(* Logix 5000 project; controller Safety vendor 1 type 14 code 86 rev 19.11; software revision 19.01; part 3 of 17 *)
(* tags used below, declared in another part *)
   MCC2_IO : UDT_CardSts[32];   // MCC2 Point I/O
   MCC2_IOSts_Flt : BOOL;   // MCC2 Point IO Module Fault ( 1= Faulted)
   MCC3_IO : UDT_CardSts[32];   // MCC3 Point I/O
   MCC3_IOSts_Flt : BOOL;   // MCC3 Point IO Module Fault ( 1= Faulted)
   MCC4_IO : UDT_CardSts[32];   // MCC4 Point I/O
   MCC4_IOSts_Flt : BOOL;   // MCC-4 Point IO Module Fault ( 1= Faulted)
   MCC5_IO : UDT_CardSts[32];   // MCC5 Point I/O
   MCC5_IOSts_Flt : BOOL;   // MCC-5 Point IO Module Fault ( 1= Faulted)
   OS11_IO : UDT_CardSts[32];   // OS11 Point I/O
   OS11_IOSts_Flt : BOOL;   // OS11 Point IO Module Fault ( 1= Faulted)
   OS13_IO : UDT_CardSts[32];   // OS13 Point I/O
   OS13_IOSts_Flt : BOOL;   // OS13 Point IO Module Fault ( 1= Faulted)
   OS14_IO : UDT_CardSts[32];   // OS14 Point I/O
   OS14_IOSts_Flt : BOOL;   // OS14 Point IO Module Fault ( 1= Faulted)
   OS15_IO : UDT_CardSts[32];   // OS15 Point I/O
   OS15_IOSts_Flt : BOOL;   // OS15 Point IO Module Fault ( 1= Faulted)
   OS16_IO : UDT_CardSts[32];   // OS16 Point I/O
   OS16_IOSts_Flt : BOOL;   // OS16 Point IO Module Fault ( 1= Faulted)
   OS1_IO : UDT_CardSts[32];   // OS1 Point I/O
   OS1_IOSts_Flt : BOOL;   // OS1 Point IO Module Fault ( 1= Faulted)
   OS2_IO : UDT_CardSts[32];   // OS2 Point I/O
   OS2_IOSts_Flt : BOOL;   // OS2 Point IO Module Fault ( 1= Faulted)
   OS3_IO : UDT_CardSts[32];   // OS3 Point I/O
   OS3_IOSts_Flt : BOOL;   // OS3 Point IO Module Fault ( 1= Faulted)
   OS4N_IO : UDT_CardSts[32];   // OS4N Point I/O
   OS4N_IOSts_Flt : BOOL;   // OS4N Point IO Module Fault ( 1= Faulted)
   OS4S_IO : UDT_CardSts[32];   // OS4S Point I/O
   OS4S_IOSts_Flt : BOOL;   // OS4S Point IO Module Fault ( 1= Faulted)
   OS5_IO : UDT_CardSts[32];   // OS5 Point I/O
   OS5_IOSts_Flt : BOOL;   // OS5 Point IO Module Fault ( 1= Faulted)
   OS6_IO : UDT_CardSts[32];   // OS6 Point I/O
   OS6_IOSts_Flt : BOOL;   // OS6 Point IO Module Fault ( 1= Faulted)
   OS8_IO : UDT_CardSts[32];   // OS8 Point I/O
   OS8_IOSts_Flt : BOOL;   // OS8 Point IO Module Fault ( 1= Faulted)
   OS9_IO : UDT_CardSts[32];   // OS9 Point I/O
   OS9_IOSts_Flt : BOOL;   // OS9 Point IO Module Fault ( 1= Faulted)
   Rem_ModFlts : DINT;   // Remote IO Comm Faults
   Sy_ClrFlt : BOOL;   // System Clear Fault
(* CardSts, continued *)

ROUTINE MCC2_IO   (* ladder *)
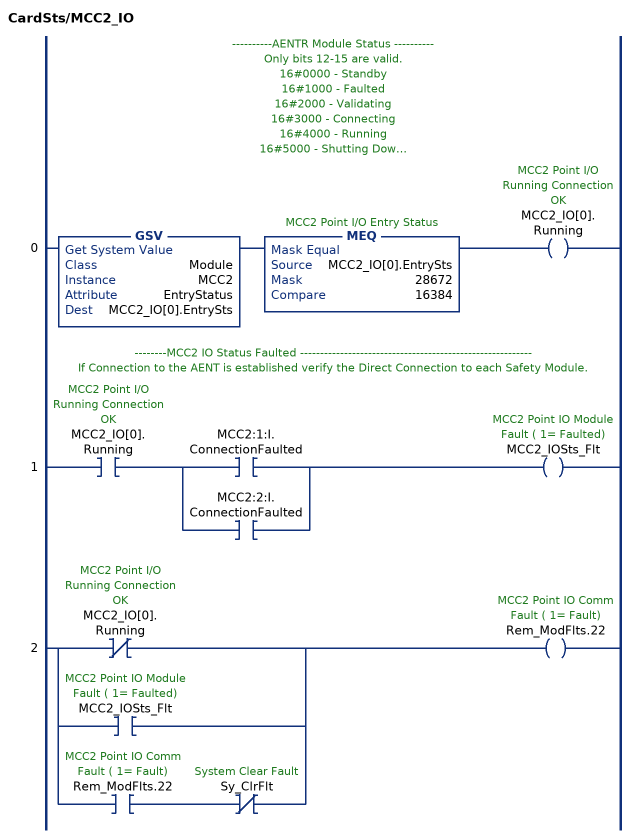
   // ----------AENTR Module Status ----------
   // Only bits 12-15 are valid.
   // 16#0000 - Standby
   // 16#1000 - Faulted
   // 16#2000 - Validating
   // 16#3000 - Connecting
   // 16#4000 - Running
   // 16#5000 - Shutting Down
   // 16#6000 - Inhibited
   // 16#7000 - Waiting
   0: GSV(Module,MCC2,EntryStatus,MCC2_IO[0].EntrySts)MEQ(MCC2_IO[0].EntrySts,28672,16384)OTE(MCC2_IO[0].Running);
   // --------MCC2 IO Status Faulted ----------------------------------------------------------
   // If Connection to the AENT is established verify the Direct Connection to each Safety Module.
   1: XIC(MCC2_IO[0].Running)[XIC(MCC2:1:I.ConnectionFaulted) ,XIC(MCC2:2:I.ConnectionFaulted) ]OTE(MCC2_IOSts_Flt);
   2: [XIO(MCC2_IO[0].Running) ,XIC(MCC2_IOSts_Flt) ,XIC(Rem_ModFlts.22) XIO(Sy_ClrFlt) ]OTE(Rem_ModFlts.22);
END_ROUTINE

ROUTINE MCC3_IO   (* ladder *)
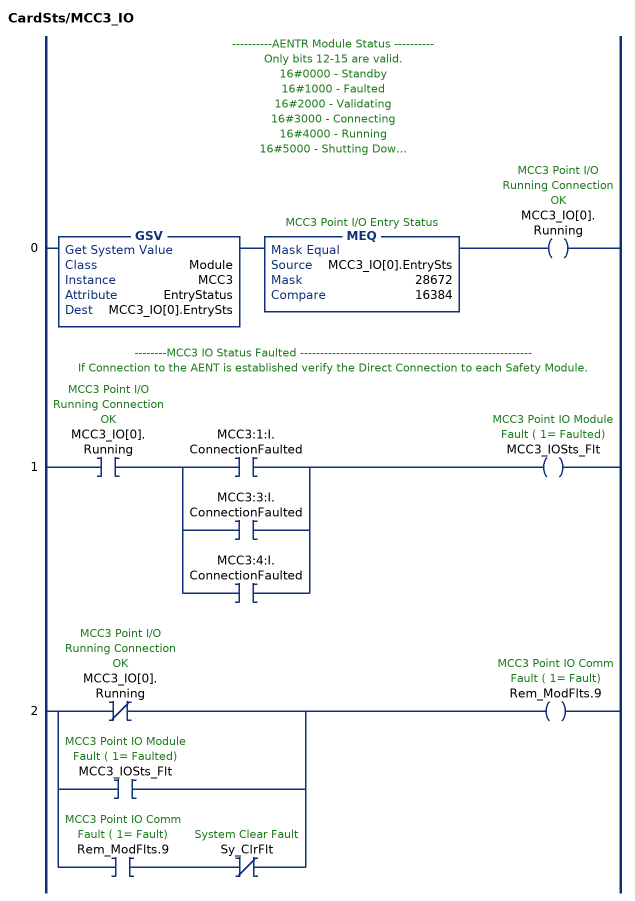
   // ----------AENTR Module Status ----------
   // Only bits 12-15 are valid.
   // 16#0000 - Standby
   // 16#1000 - Faulted
   // 16#2000 - Validating
   // 16#3000 - Connecting
   // 16#4000 - Running
   // 16#5000 - Shutting Down
   // 16#6000 - Inhibited
   // 16#7000 - Waiting
   0: GSV(Module,MCC3,EntryStatus,MCC3_IO[0].EntrySts)MEQ(MCC3_IO[0].EntrySts,28672,16384)OTE(MCC3_IO[0].Running);
   // --------MCC3 IO Status Faulted ----------------------------------------------------------
   // If Connection to the AENT is established verify the Direct Connection to each Safety Module.
   1: XIC(MCC3_IO[0].Running)[XIC(MCC3:1:I.ConnectionFaulted) ,XIC(MCC3:3:I.ConnectionFaulted) ,XIC(MCC3:4:I.ConnectionFaulted) ]OTE(MCC3_IOSts_Flt);
   2: [XIO(MCC3_IO[0].Running) ,XIC(MCC3_IOSts_Flt) ,XIC(Rem_ModFlts.9) XIO(Sy_ClrFlt) ]OTE(Rem_ModFlts.9);
END_ROUTINE

ROUTINE MCC4_IO   (* ladder *)
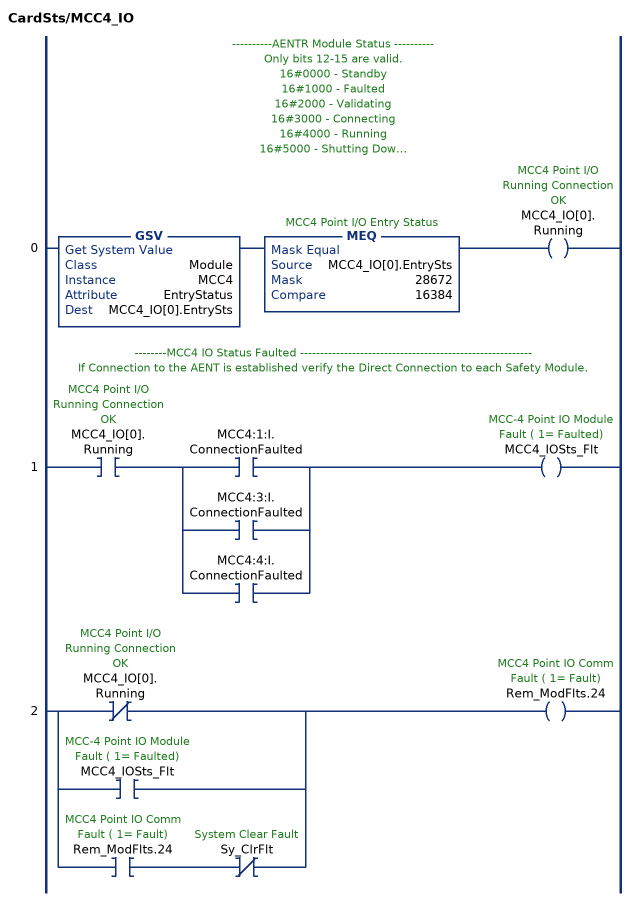
   // ----------AENTR Module Status ----------
   // Only bits 12-15 are valid.
   // 16#0000 - Standby
   // 16#1000 - Faulted
   // 16#2000 - Validating
   // 16#3000 - Connecting
   // 16#4000 - Running
   // 16#5000 - Shutting Down
   // 16#6000 - Inhibited
   // 16#7000 - Waiting
   0: GSV(Module,MCC4,EntryStatus,MCC4_IO[0].EntrySts)MEQ(MCC4_IO[0].EntrySts,28672,16384)OTE(MCC4_IO[0].Running);
   // --------MCC4 IO Status Faulted ----------------------------------------------------------
   // If Connection to the AENT is established verify the Direct Connection to each Safety Module.
   1: XIC(MCC4_IO[0].Running)[XIC(MCC4:1:I.ConnectionFaulted) ,XIC(MCC4:3:I.ConnectionFaulted) ,XIC(MCC4:4:I.ConnectionFaulted) ]OTE(MCC4_IOSts_Flt);
   2: [XIO(MCC4_IO[0].Running) ,XIC(MCC4_IOSts_Flt) ,XIC(Rem_ModFlts.24) XIO(Sy_ClrFlt) ]OTE(Rem_ModFlts.24);
END_ROUTINE

ROUTINE MCC5_IO   (* ladder *)
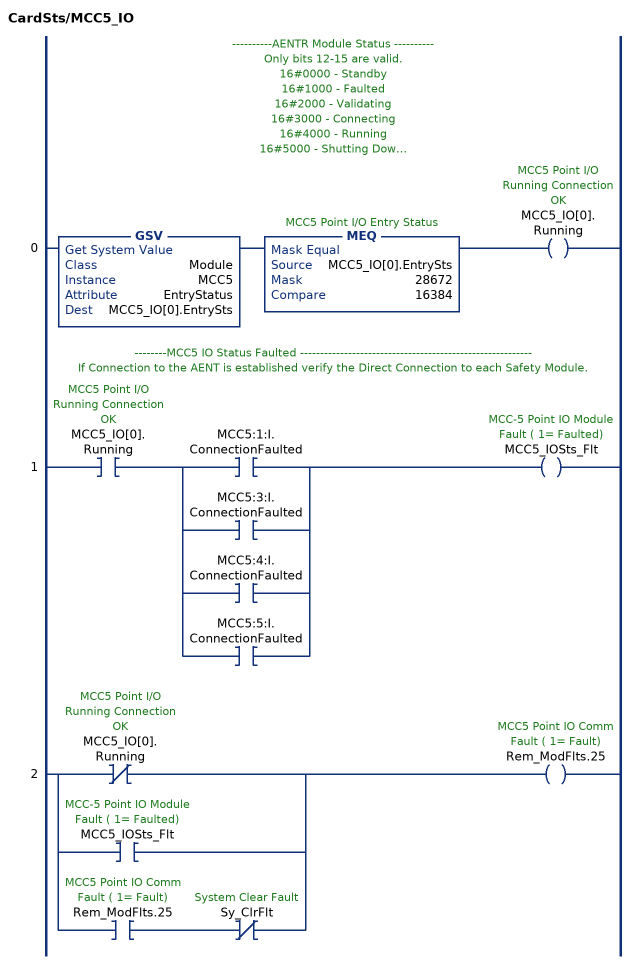
   // ----------AENTR Module Status ----------
   // Only bits 12-15 are valid.
   // 16#0000 - Standby
   // 16#1000 - Faulted
   // 16#2000 - Validating
   // 16#3000 - Connecting
   // 16#4000 - Running
   // 16#5000 - Shutting Down
   // 16#6000 - Inhibited
   // 16#7000 - Waiting
   0: GSV(Module,MCC5,EntryStatus,MCC5_IO[0].EntrySts)MEQ(MCC5_IO[0].EntrySts,28672,16384)OTE(MCC5_IO[0].Running);
   // --------MCC5 IO Status Faulted ----------------------------------------------------------
   // If Connection to the AENT is established verify the Direct Connection to each Safety Module.
   1: XIC(MCC5_IO[0].Running)[XIC(MCC5:1:I.ConnectionFaulted) ,XIC(MCC5:3:I.ConnectionFaulted) ,XIC(MCC5:4:I.ConnectionFaulted) ,XIC(MCC5:5:I.ConnectionFaulted) ]OTE(MCC5_IOSts_Flt);
   2: [XIO(MCC5_IO[0].Running) ,XIC(MCC5_IOSts_Flt) ,XIC(Rem_ModFlts.25) XIO(Sy_ClrFlt) ]OTE(Rem_ModFlts.25);
END_ROUTINE

ROUTINE OS11_IO   (* ladder *)
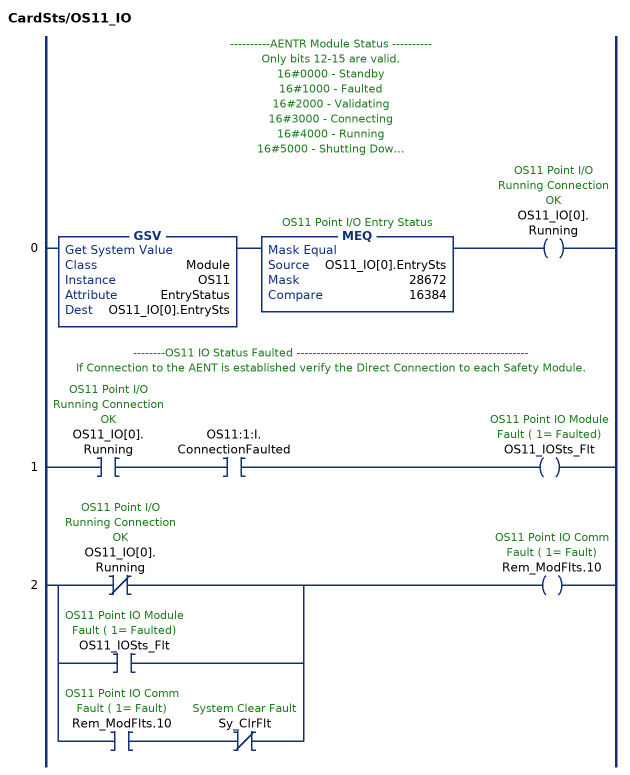
   // ----------AENTR Module Status ----------
   // Only bits 12-15 are valid.
   // 16#0000 - Standby
   // 16#1000 - Faulted
   // 16#2000 - Validating
   // 16#3000 - Connecting
   // 16#4000 - Running
   // 16#5000 - Shutting Down
   // 16#6000 - Inhibited
   // 16#7000 - Waiting
   0: GSV(Module,OS11,EntryStatus,OS11_IO[0].EntrySts)MEQ(OS11_IO[0].EntrySts,28672,16384)OTE(OS11_IO[0].Running);
   // --------OS11 IO Status Faulted ----------------------------------------------------------
   // If Connection to the AENT is established verify the Direct Connection to each Safety Module.
   1: XIC(OS11_IO[0].Running)XIC(OS11:1:I.ConnectionFaulted)OTE(OS11_IOSts_Flt);
   2: [XIO(OS11_IO[0].Running) ,XIC(OS11_IOSts_Flt) ,XIC(Rem_ModFlts.10) XIO(Sy_ClrFlt) ]OTE(Rem_ModFlts.10);
END_ROUTINE

ROUTINE OS13_IO   (* ladder *)
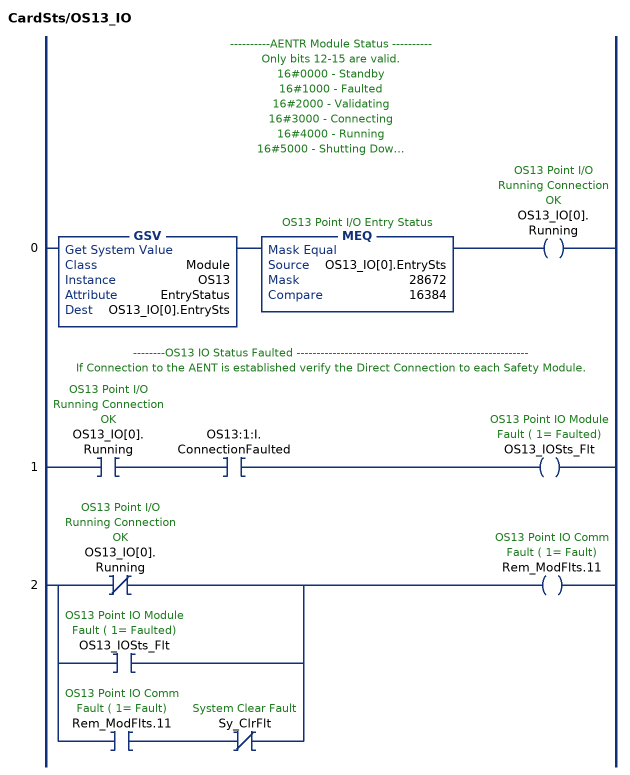
   // ----------AENTR Module Status ----------
   // Only bits 12-15 are valid.
   // 16#0000 - Standby
   // 16#1000 - Faulted
   // 16#2000 - Validating
   // 16#3000 - Connecting
   // 16#4000 - Running
   // 16#5000 - Shutting Down
   // 16#6000 - Inhibited
   // 16#7000 - Waiting
   0: GSV(Module,OS13,EntryStatus,OS13_IO[0].EntrySts)MEQ(OS13_IO[0].EntrySts,28672,16384)OTE(OS13_IO[0].Running);
   // --------OS13 IO Status Faulted ----------------------------------------------------------
   // If Connection to the AENT is established verify the Direct Connection to each Safety Module.
   1: XIC(OS13_IO[0].Running)XIC(OS13:1:I.ConnectionFaulted)OTE(OS13_IOSts_Flt);
   2: [XIO(OS13_IO[0].Running) ,XIC(OS13_IOSts_Flt) ,XIC(Rem_ModFlts.11) XIO(Sy_ClrFlt) ]OTE(Rem_ModFlts.11);
END_ROUTINE

ROUTINE OS14_IO   (* ladder *)
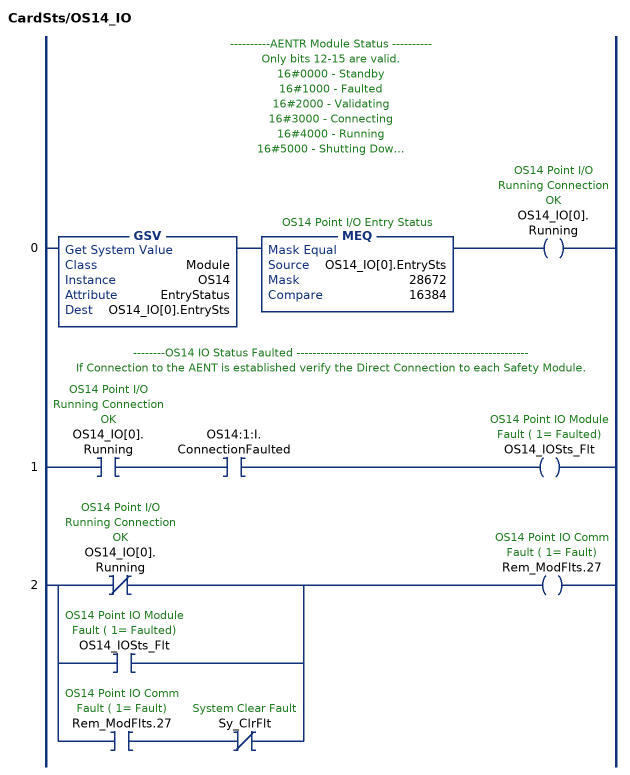
   // ----------AENTR Module Status ----------
   // Only bits 12-15 are valid.
   // 16#0000 - Standby
   // 16#1000 - Faulted
   // 16#2000 - Validating
   // 16#3000 - Connecting
   // 16#4000 - Running
   // 16#5000 - Shutting Down
   // 16#6000 - Inhibited
   // 16#7000 - Waiting
   0: GSV(Module,OS14,EntryStatus,OS14_IO[0].EntrySts)MEQ(OS14_IO[0].EntrySts,28672,16384)OTE(OS14_IO[0].Running);
   // --------OS14 IO Status Faulted ----------------------------------------------------------
   // If Connection to the AENT is established verify the Direct Connection to each Safety Module.
   1: XIC(OS14_IO[0].Running)XIC(OS14:1:I.ConnectionFaulted)OTE(OS14_IOSts_Flt);
   2: [XIO(OS14_IO[0].Running) ,XIC(OS14_IOSts_Flt) ,XIC(Rem_ModFlts.27) XIO(Sy_ClrFlt) ]OTE(Rem_ModFlts.27);
END_ROUTINE

ROUTINE OS15_IO   (* ladder *)
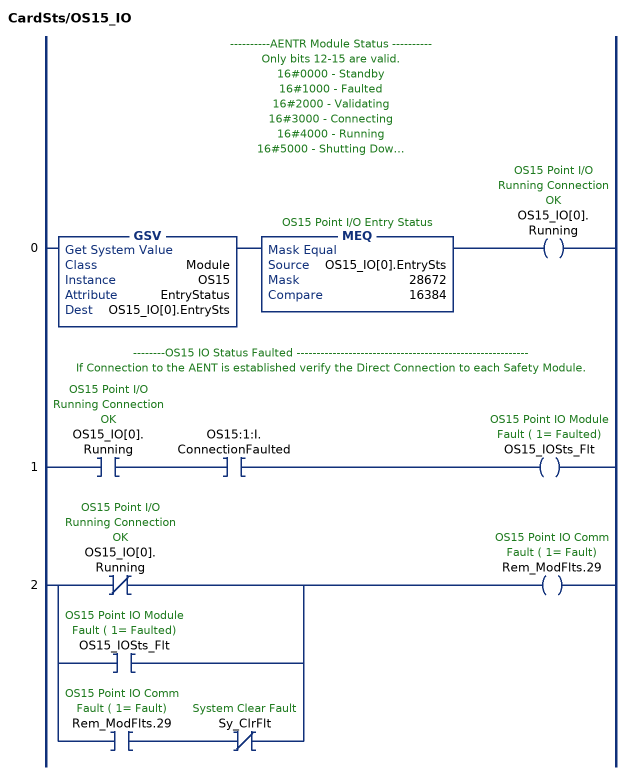
   // ----------AENTR Module Status ----------
   // Only bits 12-15 are valid.
   // 16#0000 - Standby
   // 16#1000 - Faulted
   // 16#2000 - Validating
   // 16#3000 - Connecting
   // 16#4000 - Running
   // 16#5000 - Shutting Down
   // 16#6000 - Inhibited
   // 16#7000 - Waiting
   0: GSV(Module,OS15,EntryStatus,OS15_IO[0].EntrySts)MEQ(OS15_IO[0].EntrySts,28672,16384)OTE(OS15_IO[0].Running);
   // --------OS15 IO Status Faulted ----------------------------------------------------------
   // If Connection to the AENT is established verify the Direct Connection to each Safety Module.
   1: XIC(OS15_IO[0].Running)XIC(OS15:1:I.ConnectionFaulted)OTE(OS15_IOSts_Flt);
   2: [XIO(OS15_IO[0].Running) ,XIC(OS15_IOSts_Flt) ,XIC(Rem_ModFlts.29) XIO(Sy_ClrFlt) ]OTE(Rem_ModFlts.29);
END_ROUTINE

ROUTINE OS16_IO   (* ladder *)
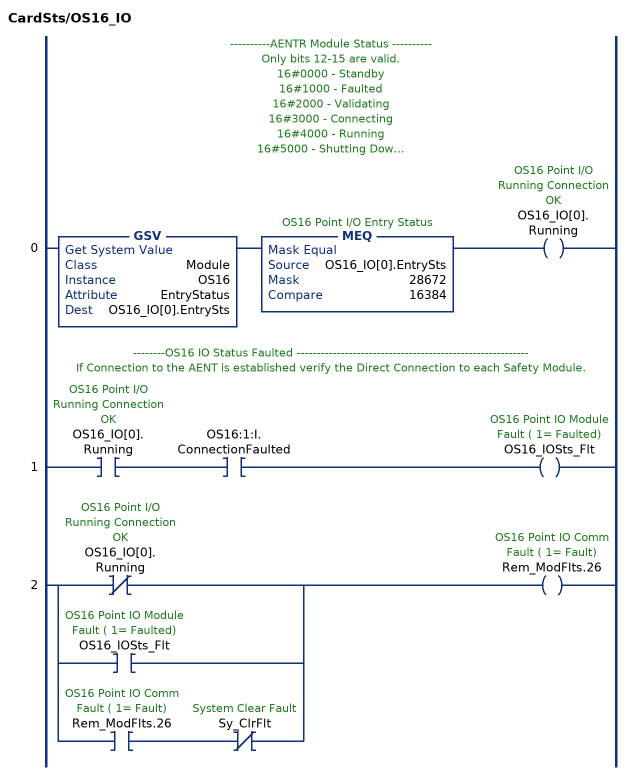
   // ----------AENTR Module Status ----------
   // Only bits 12-15 are valid.
   // 16#0000 - Standby
   // 16#1000 - Faulted
   // 16#2000 - Validating
   // 16#3000 - Connecting
   // 16#4000 - Running
   // 16#5000 - Shutting Down
   // 16#6000 - Inhibited
   // 16#7000 - Waiting
   0: GSV(Module,OS16,EntryStatus,OS16_IO[0].EntrySts)MEQ(OS16_IO[0].EntrySts,28672,16384)OTE(OS16_IO[0].Running);
   // --------OS16 IO Status Faulted ----------------------------------------------------------
   // If Connection to the AENT is established verify the Direct Connection to each Safety Module.
   1: XIC(OS16_IO[0].Running)XIC(OS16:1:I.ConnectionFaulted)OTE(OS16_IOSts_Flt);
   2: [XIO(OS16_IO[0].Running) ,XIC(OS16_IOSts_Flt) ,XIC(Rem_ModFlts.26) XIO(Sy_ClrFlt) ]OTE(Rem_ModFlts.26);
END_ROUTINE

ROUTINE OS1_IO   (* ladder *)
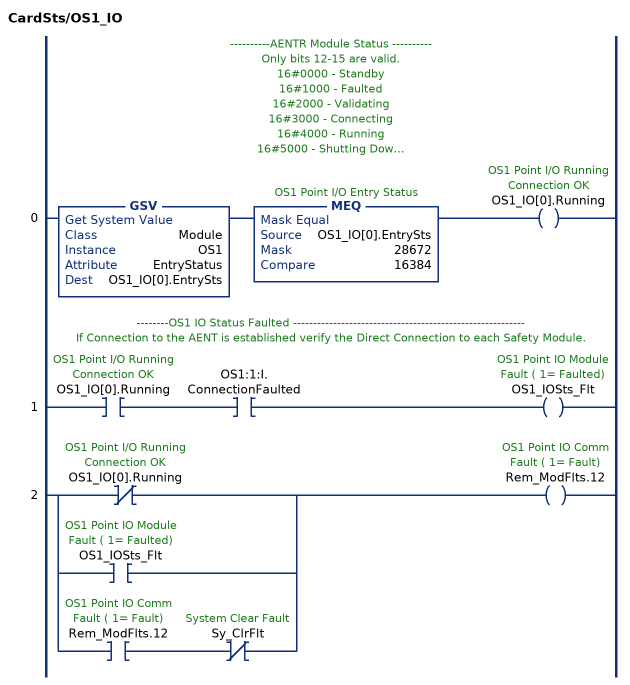
   // ----------AENTR Module Status ----------
   // Only bits 12-15 are valid.
   // 16#0000 - Standby
   // 16#1000 - Faulted
   // 16#2000 - Validating
   // 16#3000 - Connecting
   // 16#4000 - Running
   // 16#5000 - Shutting Down
   // 16#6000 - Inhibited
   // 16#7000 - Waiting
   0: GSV(Module,OS1,EntryStatus,OS1_IO[0].EntrySts)MEQ(OS1_IO[0].EntrySts,28672,16384)OTE(OS1_IO[0].Running);
   // --------OS1 IO Status Faulted ----------------------------------------------------------
   // If Connection to the AENT is established verify the Direct Connection to each Safety Module.
   1: XIC(OS1_IO[0].Running)XIC(OS1:1:I.ConnectionFaulted)OTE(OS1_IOSts_Flt);
   2: [XIO(OS1_IO[0].Running) ,XIC(OS1_IOSts_Flt) ,XIC(Rem_ModFlts.12) XIO(Sy_ClrFlt) ]OTE(Rem_ModFlts.12);
END_ROUTINE

ROUTINE OS2_IO   (* ladder *)
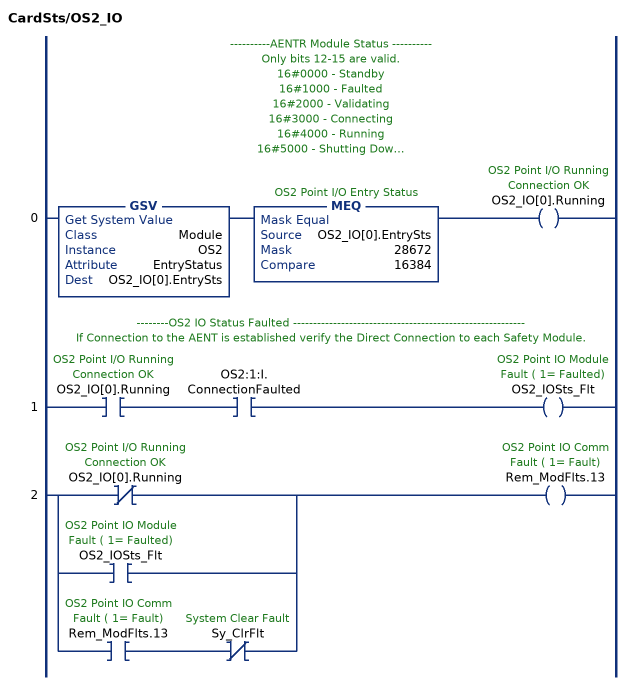
   // ----------AENTR Module Status ----------
   // Only bits 12-15 are valid.
   // 16#0000 - Standby
   // 16#1000 - Faulted
   // 16#2000 - Validating
   // 16#3000 - Connecting
   // 16#4000 - Running
   // 16#5000 - Shutting Down
   // 16#6000 - Inhibited
   // 16#7000 - Waiting
   0: GSV(Module,OS2,EntryStatus,OS2_IO[0].EntrySts)MEQ(OS2_IO[0].EntrySts,28672,16384)OTE(OS2_IO[0].Running);
   // --------OS2 IO Status Faulted ----------------------------------------------------------
   // If Connection to the AENT is established verify the Direct Connection to each Safety Module.
   1: XIC(OS2_IO[0].Running)XIC(OS2:1:I.ConnectionFaulted)OTE(OS2_IOSts_Flt);
   2: [XIO(OS2_IO[0].Running) ,XIC(OS2_IOSts_Flt) ,XIC(Rem_ModFlts.13) XIO(Sy_ClrFlt) ]OTE(Rem_ModFlts.13);
END_ROUTINE

ROUTINE OS3_IO   (* ladder *)
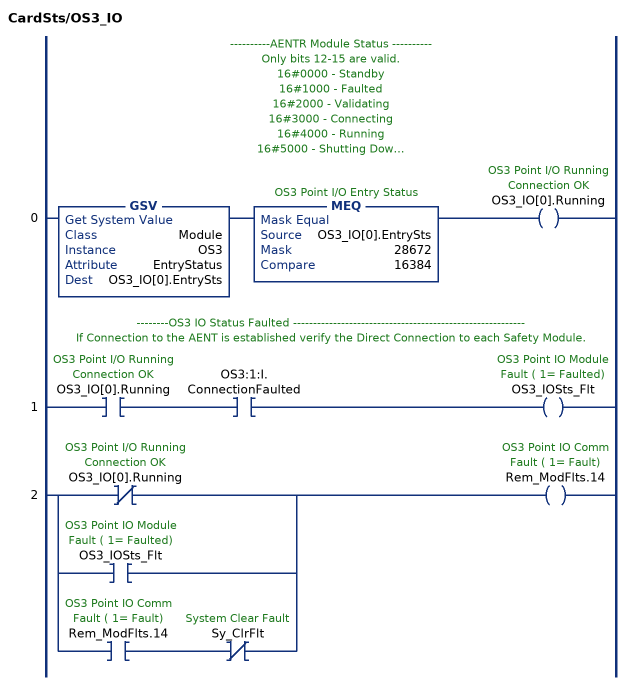
   // ----------AENTR Module Status ----------
   // Only bits 12-15 are valid.
   // 16#0000 - Standby
   // 16#1000 - Faulted
   // 16#2000 - Validating
   // 16#3000 - Connecting
   // 16#4000 - Running
   // 16#5000 - Shutting Down
   // 16#6000 - Inhibited
   // 16#7000 - Waiting
   0: GSV(Module,OS3,EntryStatus,OS3_IO[0].EntrySts)MEQ(OS3_IO[0].EntrySts,28672,16384)OTE(OS3_IO[0].Running);
   // --------OS3 IO Status Faulted ----------------------------------------------------------
   // If Connection to the AENT is established verify the Direct Connection to each Safety Module.
   1: XIC(OS3_IO[0].Running)XIC(OS3:1:I.ConnectionFaulted)OTE(OS3_IOSts_Flt);
   2: [XIO(OS3_IO[0].Running) ,XIC(OS3_IOSts_Flt) ,XIC(Rem_ModFlts.14) XIO(Sy_ClrFlt) ]OTE(Rem_ModFlts.14);
END_ROUTINE

ROUTINE OS4N_IO   (* ladder *)
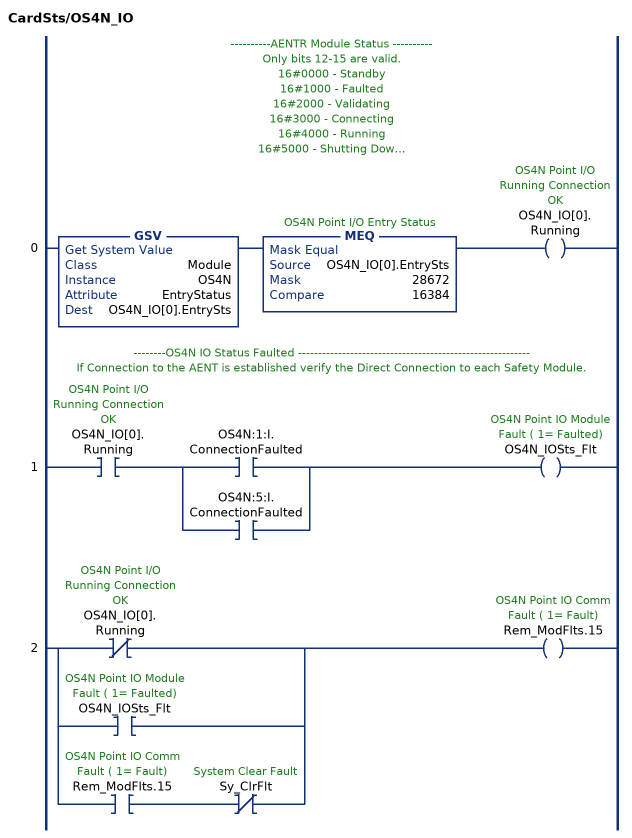
   // ----------AENTR Module Status ----------
   // Only bits 12-15 are valid.
   // 16#0000 - Standby
   // 16#1000 - Faulted
   // 16#2000 - Validating
   // 16#3000 - Connecting
   // 16#4000 - Running
   // 16#5000 - Shutting Down
   // 16#6000 - Inhibited
   // 16#7000 - Waiting
   0: GSV(Module,OS4N,EntryStatus,OS4N_IO[0].EntrySts)MEQ(OS4N_IO[0].EntrySts,28672,16384)OTE(OS4N_IO[0].Running);
   // --------OS4N IO Status Faulted ----------------------------------------------------------
   // If Connection to the AENT is established verify the Direct Connection to each Safety Module.
   1: XIC(OS4N_IO[0].Running)[XIC(OS4N:1:I.ConnectionFaulted) ,XIC(OS4N:5:I.ConnectionFaulted) ]OTE(OS4N_IOSts_Flt);
   2: [XIO(OS4N_IO[0].Running) ,XIC(OS4N_IOSts_Flt) ,XIC(Rem_ModFlts.15) XIO(Sy_ClrFlt) ]OTE(Rem_ModFlts.15);
END_ROUTINE

ROUTINE OS4S_IO   (* ladder *)
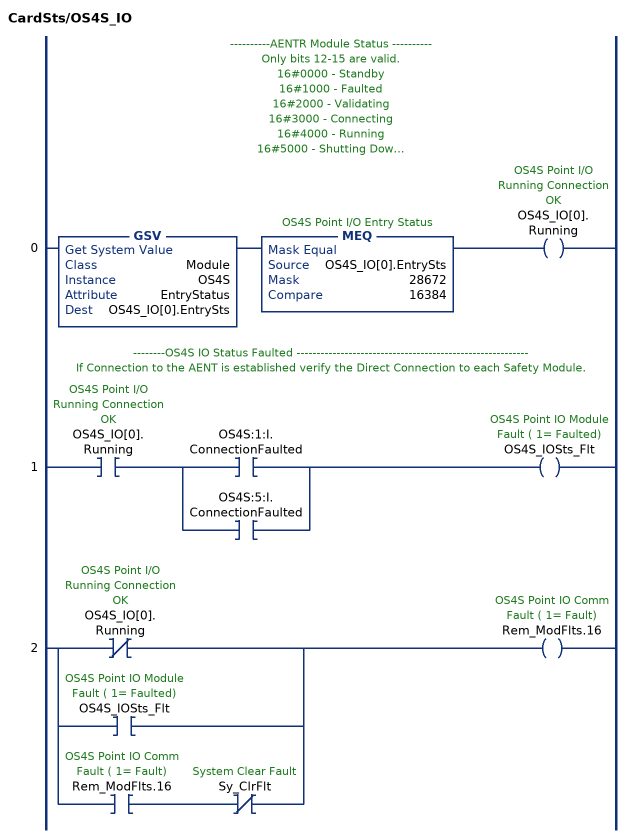
   // ----------AENTR Module Status ----------
   // Only bits 12-15 are valid.
   // 16#0000 - Standby
   // 16#1000 - Faulted
   // 16#2000 - Validating
   // 16#3000 - Connecting
   // 16#4000 - Running
   // 16#5000 - Shutting Down
   // 16#6000 - Inhibited
   // 16#7000 - Waiting
   0: GSV(Module,OS4S,EntryStatus,OS4S_IO[0].EntrySts)MEQ(OS4S_IO[0].EntrySts,28672,16384)OTE(OS4S_IO[0].Running);
   // --------OS4S IO Status Faulted ----------------------------------------------------------
   // If Connection to the AENT is established verify the Direct Connection to each Safety Module.
   1: XIC(OS4S_IO[0].Running)[XIC(OS4S:1:I.ConnectionFaulted) ,XIC(OS4S:5:I.ConnectionFaulted) ]OTE(OS4S_IOSts_Flt);
   2: [XIO(OS4S_IO[0].Running) ,XIC(OS4S_IOSts_Flt) ,XIC(Rem_ModFlts.16) XIO(Sy_ClrFlt) ]OTE(Rem_ModFlts.16);
END_ROUTINE

ROUTINE OS5_IO   (* ladder *)
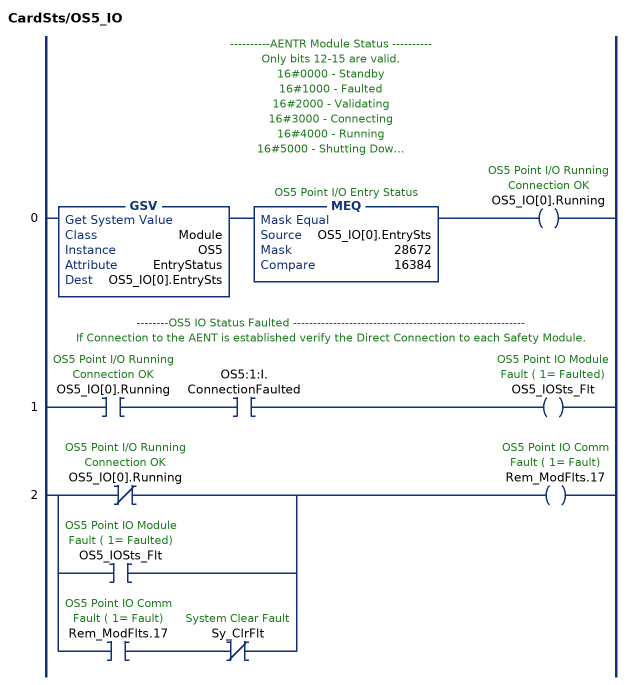
   // ----------AENTR Module Status ----------
   // Only bits 12-15 are valid.
   // 16#0000 - Standby
   // 16#1000 - Faulted
   // 16#2000 - Validating
   // 16#3000 - Connecting
   // 16#4000 - Running
   // 16#5000 - Shutting Down
   // 16#6000 - Inhibited
   // 16#7000 - Waiting
   0: GSV(Module,OS5,EntryStatus,OS5_IO[0].EntrySts)MEQ(OS5_IO[0].EntrySts,28672,16384)OTE(OS5_IO[0].Running);
   // --------OS5 IO Status Faulted ----------------------------------------------------------
   // If Connection to the AENT is established verify the Direct Connection to each Safety Module.
   1: XIC(OS5_IO[0].Running)XIC(OS5:1:I.ConnectionFaulted)OTE(OS5_IOSts_Flt);
   2: [XIO(OS5_IO[0].Running) ,XIC(OS5_IOSts_Flt) ,XIC(Rem_ModFlts.17) XIO(Sy_ClrFlt) ]OTE(Rem_ModFlts.17);
END_ROUTINE

ROUTINE OS6_IO   (* ladder *)
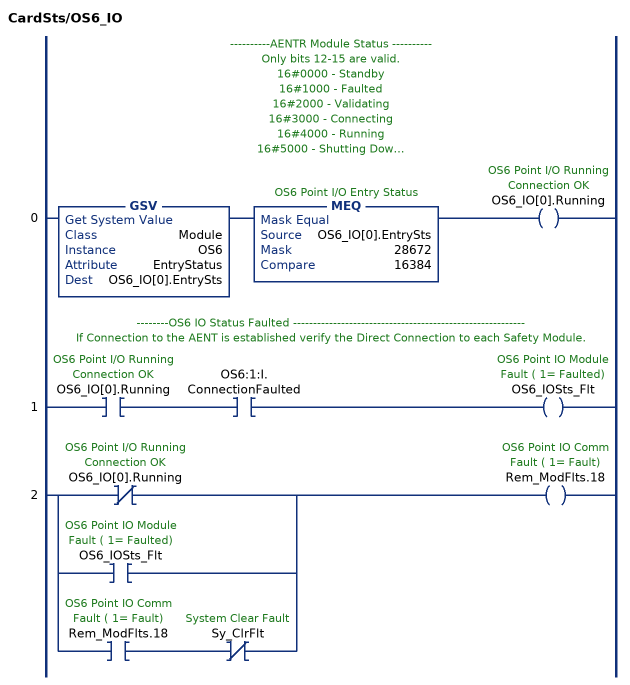
   // ----------AENTR Module Status ----------
   // Only bits 12-15 are valid.
   // 16#0000 - Standby
   // 16#1000 - Faulted
   // 16#2000 - Validating
   // 16#3000 - Connecting
   // 16#4000 - Running
   // 16#5000 - Shutting Down
   // 16#6000 - Inhibited
   // 16#7000 - Waiting
   0: GSV(Module,OS6,EntryStatus,OS6_IO[0].EntrySts)MEQ(OS6_IO[0].EntrySts,28672,16384)OTE(OS6_IO[0].Running);
   // --------OS6 IO Status Faulted ----------------------------------------------------------
   // If Connection to the AENT is established verify the Direct Connection to each Safety Module.
   1: XIC(OS6_IO[0].Running)XIC(OS6:1:I.ConnectionFaulted)OTE(OS6_IOSts_Flt);
   2: [XIO(OS6_IO[0].Running) ,XIC(OS6_IOSts_Flt) ,XIC(Rem_ModFlts.18) XIO(Sy_ClrFlt) ]OTE(Rem_ModFlts.18);
END_ROUTINE

ROUTINE OS8_IO   (* ladder *)
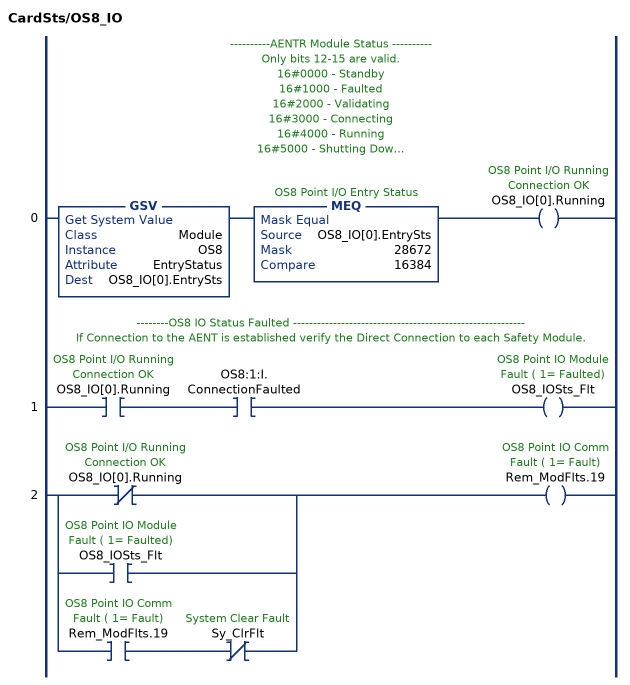
   // ----------AENTR Module Status ----------
   // Only bits 12-15 are valid.
   // 16#0000 - Standby
   // 16#1000 - Faulted
   // 16#2000 - Validating
   // 16#3000 - Connecting
   // 16#4000 - Running
   // 16#5000 - Shutting Down
   // 16#6000 - Inhibited
   // 16#7000 - Waiting
   0: GSV(Module,OS8,EntryStatus,OS8_IO[0].EntrySts)MEQ(OS8_IO[0].EntrySts,28672,16384)OTE(OS8_IO[0].Running);
   // --------OS8 IO Status Faulted ----------------------------------------------------------
   // If Connection to the AENT is established verify the Direct Connection to each Safety Module.
   1: XIC(OS8_IO[0].Running)XIC(OS8:1:I.ConnectionFaulted)OTE(OS8_IOSts_Flt);
   2: [XIO(OS8_IO[0].Running) ,XIC(OS8_IOSts_Flt) ,XIC(Rem_ModFlts.19) XIO(Sy_ClrFlt) ]OTE(Rem_ModFlts.19);
END_ROUTINE

ROUTINE OS9_IO   (* ladder *)
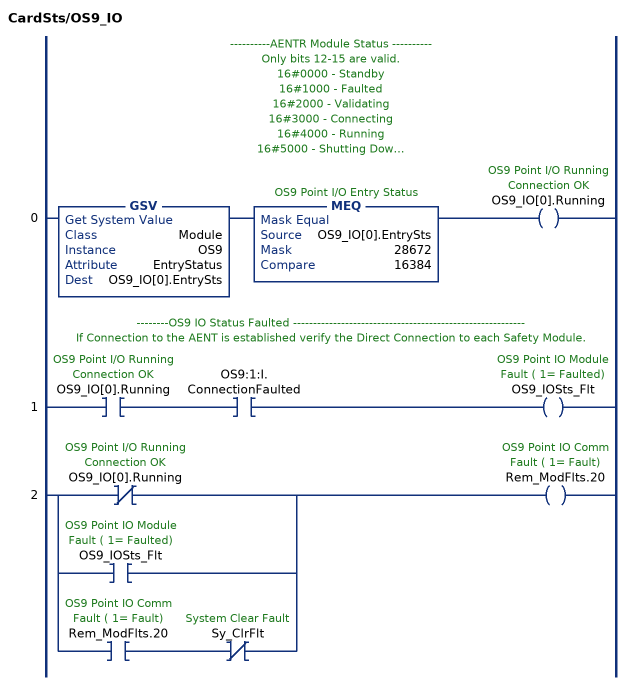
   // ----------AENTR Module Status ----------
   // Only bits 12-15 are valid.
   // 16#0000 - Standby
   // 16#1000 - Faulted
   // 16#2000 - Validating
   // 16#3000 - Connecting
   // 16#4000 - Running
   // 16#5000 - Shutting Down
   // 16#6000 - Inhibited
   // 16#7000 - Waiting
   0: GSV(Module,OS9,EntryStatus,OS9_IO[0].EntrySts)MEQ(OS9_IO[0].EntrySts,28672,16384)OTE(OS9_IO[0].Running);
   // --------OS9 IO Status Faulted ----------------------------------------------------------
   // If Connection to the AENT is established verify the Direct Connection to each Safety Module.
   1: XIC(OS9_IO[0].Running)XIC(OS9:1:I.ConnectionFaulted)OTE(OS9_IOSts_Flt);
   2: [XIO(OS9_IO[0].Running) ,XIC(OS9_IOSts_Flt) ,XIC(Rem_ModFlts.20) XIO(Sy_ClrFlt) ]OTE(Rem_ModFlts.20);
END_ROUTINE
